{attribute 'GeneratedUsingTerminal: EM3701-0000-0016'}
{attribute addProperty BoxType "EM3701-0000-0016"}
{attribute addProperty Id "AI_InputsAT %I*AI_Inputs_5AF6604E8WcStateAT %I*WcState_9091E0EB2InfoDataAT %I*InfoData_32EB74EA10"}
{attribute addProperty CRC "2869773981"}
{attribute addProperty Size "20"}
TYPE EM3701_AB0D469D EXTENDS EtcSlaveTerminalBase_947E5A46 :
STRUCT
	{attribute addProperty Name "AI_Inputs"}
	AI_Inputs : AI_Inputs_5AF6604E;
	{attribute addProperty Name "WcState"}
	WcState : WcState_9091E0EB;
	{attribute addProperty Name "InfoData"}
	InfoData : InfoData_32EB74EA;
END_STRUCT
END_TYPE

(* stored: Version 1.2.0.0, ProductVersion 3.1.4024.9
   DUT EM3701_AB0D469D: Id {d3cafc93-c6cc-4b50-be49-16c697cc452f} *)
